(* IEC 61131-3 sources: Moonplc/examples, 4 files *)

(* ---- 01_motor_start_stop.st ---- *)
(* 工业经典案例 01: 电机自锁起保停控制系统 *)
PROGRAM MotorStartStop
VAR
  Start_Btn AT %IX0.0 : BOOL := FALSE; (* 启动按钮 (常开) *)
  Stop_Btn  AT %IX0.1 : BOOL := FALSE; (* 停止按钮 (常闭输入) *)
  Motor_Run AT %QX0.0 : BOOL := FALSE; (* 电机接触器输出 *)
  Fault_Led AT %QX0.1 : BOOL := FALSE; (* 故障指示灯 *)
END_VAR

(* 梯形图等价自锁逻辑 *)
Motor_Run := (Start_Btn OR Motor_Run) AND NOT Stop_Btn;
END_PROGRAM

(* ---- 02_traffic_light.st ---- *)
(* 工业经典案例 02: 道路路口智能交通信号灯顺序控制 *)
PROGRAM TrafficLightControl
VAR
  Car_Present AT %IX0.0 : BOOL := FALSE; (* 地感线圈车辆感应 *)
  Pedestrian  AT %IX0.1 : BOOL := FALSE; (* 行人过街请求按钮 *)
  Light_Red   AT %QX0.0 : BOOL := TRUE;  (* 红灯输出 *)
  Light_Green AT %QX0.1 : BOOL := FALSE; (* 绿灯输出 *)
  Light_Amber AT %QX0.2 : BOOL := FALSE; (* 黄灯输出 *)
  Timer_Pass  : TON;                     (* 通行定时器 *)
END_VAR

(* 交通控制逻辑 *)
IF Car_Present OR Pedestrian THEN
  Light_Red   := FALSE;
  Light_Green := TRUE;
  Timer_Pass(IN := TRUE, PT := T#3000ms);

  IF Timer_Pass.Q THEN
    Light_Green := FALSE;
    Light_Amber := TRUE;
  END_IF;
ELSE
  Light_Red   := TRUE;
  Light_Green := FALSE;
  Light_Amber := FALSE;
  Timer_Pass(IN := FALSE, PT := T#3000ms);
END_IF;
END_PROGRAM

(* ---- 03_conveyor_sorting.st ---- *)
(* 工业经典案例 03: 自动化传送带物料感应与气动推杆分拣系统 *)
PROGRAM ConveyorSorting
VAR
  Sensor_Item AT %IX0.0 : BOOL := FALSE; (* 光电检测传感器 *)
  Belt_Motor  AT %QX0.0 : BOOL := TRUE;  (* 主传送带电机 *)
  Piston_Push AT %QX0.1 : BOOL := FALSE; (* 气动推杆阀门 *)
  Item_Count  : INT := 0;                (* 物料累计计数 *)
  Piston_Timer : TP;                     (* 气缸脉冲定时器 *)
END_VAR

(* 检测到物料时触发气动推杆脉冲 *)
Piston_Timer(IN := Sensor_Item, PT := T#500ms);
Piston_Push := Piston_Timer.Q;

IF Sensor_Item THEN
  Item_Count := Item_Count + 1;
END_IF;
END_PROGRAM

(* ---- 05_pid_temperature_tank.st ---- *)
(* 工业经典案例 05: 水箱恒温闭环 PID 控制系统 *)
PROGRAM TemperatureControl
VAR
  Temp_SP       : REAL := 65.0;            (* 目标设定温度: 65.0°C *)
  Temp_PV       AT %IW0 : REAL := 20.0;    (* 现场 PT100 传感器采集温度 *)
  Heater_Output AT %QW0 : REAL := 0.0;     (* 可控硅加热器输出功率 (0~100%) *)
  Cooling_Valve AT %QX0.0 : BOOL := FALSE; (* 应急冷却电磁阀 *)
  Temp_Alarm    AT %QX0.1 : BOOL := FALSE; (* 超温上限报警灯 *)
END_VAR

(* 超温安全连锁保护 *)
IF Temp_PV > 80.0 THEN
  Temp_Alarm := TRUE;
  Cooling_Valve := TRUE;
  Heater_Output := 0.0;
ELSE
  Temp_Alarm := FALSE;
  Cooling_Valve := FALSE;
END_IF;
END_PROGRAM
